# EPICS substitutions: db/Beckhoff_3XXX/ecmcEP3751-0160.substitutions
file "ecmc_analogInput-chX.template"
{
  pattern {CH_ID, sourceName, KEY, ESLO, EOFF, PREC, EGU}
          {X, accelerationActual, AcclAct, "${_ESLO=0.001}", "${_EOFF=0}", "${_PREC=3}", "${_EGU=g}"}
          {Y, accelerationActual, AcclAct, "${_ESLO=0.001}", "${_EOFF=0}", "${_PREC=3}", "${_EGU=g}"}
          {Z, accelerationActual, AcclAct, "${_ESLO=0.001}", "${_EOFF=0}", "${_PREC=3}", "${_EGU=g}"}
          {'', temperature, Temp, "${_ESLO=1.0}", "${_EOFF=0}", "${_PREC=0}", "${_EGU=degC}"}
}
